// Brake faults section
// Brake cam switch monitoring
TON_1(IN := Lh_off AND Lh_rubbing AND Mode.Brake_maintenance, PT := t#200ms); // TON
TON_2(IN := Rh_off AND Rh_rubbing AND Mode.Brake_maintenance, PT := t#200ms); // TON
cs_Lh_off_before_rubbing := TON_1.Q;
cs_Rh_off_before_rubbing := TON_2.Q;
TON_3(IN := Lh_on AND Lh_rubbing AND Mode.Brake_maintenance, PT := t#200ms); // TON
TON_4(IN := Rh_on AND Rh_rubbing AND Mode.Brake_maintenance, PT := t#200ms); // TON
cs_Lh_on_and_rubbing := TON_3.Q;
cs_Rh_on_and_rubbing := TON_4.Q;
TON_5(IN := Lh_wear AND Lh_on AND Mode.Brake_maintenance, PT := t#200ms); // TON
TON_6(IN := Rh_wear AND Rh_on AND Mode.Brake_maintenance, PT := t#200ms); // TON
cs_Lh_wear_before_on := TON_5.Q;
cs_Rh_wear_before_on := TON_6.Q;
TON_7(IN := Lh_on AND Lh_off AND Mode.Brake_maintenance, PT := t#200ms); // TON
TON_8(IN := Rh_on AND Rh_off AND Mode.Brake_maintenance, PT := t#200ms); // TON
cs_Lh_on_and_off := TON_7.Q;
cs_Rh_on_and_off := TON_8.Q;
TON_9(IN := Lever_on AND Lever_off AND Mode.Brake_maintenance, PT := t#200ms); // TON
TON_10(IN := Lever_on AND Lever_fully_off AND Mode.Brake_maintenance, PT := t#200ms); // TON
cs_Lever_off_and_on := TON_9.Q;
cs_Lever_fully_off_and_on := TON_10.Q;
// Brake lever monitoring
TON_11(IN := Lever_fully_off AND Mode.Manual OR Mode.Auto_go, PT := Off_time); // TON
TON_12(IN := TON_11.Q AND NOT Lh_off AND NOT Trail_brakes AND Clutch.Lh_in AND NOT Lh_test AND Safety.Sc1 AND NOT Mode.Brake_maintenance, PT := t#3s); // TON
cs_Lh_not_fully_off := TON_12.Q;
TON_13(IN := Lever_fully_off AND Mode.Manual OR Mode.Auto_go, PT := Off_time); // TON
TON_14(IN := TON_13.Q AND NOT Rh_off AND NOT Trail_brakes AND Clutch.Rh_in AND NOT Rh_test AND Safety.Sc1 AND NOT Mode.Brake_maintenance, PT := t#3s); // TON
cs_Rh_not_fully_off := TON_14.Q;
TON_15(IN := Lever_on, PT := On_time); // TON
tr_Lh_not_on := TON_15.Q AND NOT Lh_on AND NOT Mode.Brake_maintenance;
// Brake rubbing trips
TON_16(IN := (ABS(Lh_speed)) > Rubbing_speed AND NOT Lh_rubbing AND Safety.Sc1 AND _w1, PT := Rubbing_time); // TON
tr_Lh_rubbing_trip := TON_16.Q;
_w1 := (ABS(Lh_speed)) > 1200 OR TON_17.Q;
TON_17(IN := NOT Trail_brakes, PT := t#1s); // TON
_w3 := TON_17.Q OR _w2;
_w2 := (ABS(Rh_speed)) > 1200;
TON_16(IN := _w3 AND _w4 AND NOT Rh_rubbing AND Safety.Sc1, PT := Rubbing_time); // TON
_w4 := (ABS(Rh_speed)) > Rubbing_speed;
tr_Rh_rubbing_trip := TON_16.Q;
// Brake maintenance trips
tr_No_brake_on_in_maint := Maintenance AND NOT Lh_on AND NOT Rh_on;
tr_Movement_in_maint := Maintenance AND Movement_detect;
tr_Maint_switch_on := NOT (Lh_on OR Rh_on) AND Maintenance_switch;
END_METHOD

END_FUNCTION_BLOCK

// ---- POUs/FBs/FB_Clutch.TcPOU
FUNCTION_BLOCK FB_Clutch
VAR_INPUT
	Lh_in:BOOL; (*Left hand clutch in switch*)
	Lh_out:BOOL; (*Left hand clutch out switch*)
	Rh_in:BOOL; (*Right hand clutch in switch*)
	Rh_out:BOOL; (*Right hand clutch out switch*)
	Lh_movement:BOOL; (*Movement on left hand drum*)
	Rh_movement:BOOL; (*Movement on right hand drum*)
	Lh_raw_depth:DINT; (*Left conveyance raw depth*)
	Rh_raw_depth:DINT; (*Right conveyance raw depth*)
	Allowed_travel_when_out:DINT; (*Amount of travel allowed while engaging/disengaging a clutch*)
END_VAR
VAR_OUTPUT
	tr_Lh_in_and_out:BOOL; (*Left hand clutch in and out switches both energised*)
	tr_Rh_in_and_out:BOOL; (*Right hand clutch in and out switches both energised*)
	tr_Lh_out_movement:BOOL; (*Movement was detected on the left hand drum when the left clutch was out*)
	tr_Rh_out_movement:BOOL; (*Movement was detected on the right hand drum when the right clutch was out*)
	tr_Lh_not_in_movement:BOOL; (*Movement was detected on the left hand drum when the left clutch was not in*)
	tr_Rh_not_in_movement:BOOL; (*Movement was detected on the right hand drum when the right clutch was not in*)
	cs_Too_much_travel_clutching:BOOL; (*There was too much drum travel while engaging/disengaging a clutch*)
	hmi_Status:WORD; (*Status bits for HMI*)
END_VAR
VAR
	TON_0: TON;
	TON_1: TON;
	TON_2: TON;
	TON_3: TON;
	Lh_start_depth: DINT;
	RS_0: RS;
	Rh_start_depth: DINT;
	RS_1: RS;
END_VAR

M_Clutch_data();
M_Clutch_faults();
M_Too_much_travel();

METHOD M_Clutch_data
VAR_INPUT
END_VAR

VAR
	BIT_TO_WORD_V0_0: FB_BIT_TO_WORD_V0;
END_VAR
// Clutch data section
Clutch.Lh_in := Lh_in;
Clutch.Rh_in := Rh_in;
Clutch.Lh_out := Lh_out;
Clutch.Rh_out := Rh_out;
Clutch.Single_drum := Lh_out OR Rh_out;
BIT_TO_WORD_V0_0(bit0 := Lh_in, bit1 := Lh_out, bit2 := Rh_in, bit3 := Rh_out, bit4 := Clutch.Single_drum); // FB_BIT_TO_WORD_V0
hmi_Status := BIT_TO_WORD_V0_0.Word_out;
END_METHOD

METHOD M_Clutch_faults
VAR_INPUT
END_VAR
// Clutch faults section
tr_Lh_in_and_out := Lh_in AND Lh_out;
tr_Rh_in_and_out := Rh_in AND Rh_out;
TON_0(IN := Lh_movement AND Lh_out, PT := t#50ms); // TON
TON_2(IN := Rh_movement AND Rh_out, PT := t#50ms); // TON
tr_Lh_out_movement := TON_0.Q;
tr_Rh_out_movement := TON_2.Q;
TON_1(IN := Lh_movement AND Lh_in, PT := t#50ms); // TON
TON_3(IN := Rh_movement AND Rh_in, PT := t#50ms); // TON
tr_Lh_not_in_movement := TON_1.Q;
tr_Rh_not_in_movement := TON_3.Q;
END_METHOD

METHOD M_Too_much_travel
VAR_INPUT
END_VAR
VAR_INST // added by the converter: edge detectors and wires of the graphical bodies
    _w1, _w3 : ANY;
    _w2, _w4 : DINT;
END_VAR
// Too much travel section
RS_0(SET := ABS(Lh_raw_depth - Lh_start_depth) > Allowed_travel_when_out, RESET1 := _w1); // RS
cs_Too_much_travel_clutching := RS_0.Q1 OR RS_1.Q1;
_w1 := Rh_in OR Rh_out OR Safety.Reset_interlocks;
IF _w1 THEN _w2 := Lh_raw_depth; END_IF
Lh_start_depth := _w2;
RS_1(SET := ABS(Rh_raw_depth - Rh_start_depth) > Allowed_travel_when_out, RESET1 := _w3); // RS
_w3 := Lh_in OR Lh_out OR Safety.Reset_interlocks;
IF _w3 THEN _w4 := Rh_raw_depth; END_IF
Rh_start_depth := _w4;
END_METHOD

END_FUNCTION_BLOCK

// ---- POUs/FBs/FB_Disc_brake.TcPOU
FUNCTION_BLOCK FB_Disc_brake
VAR_INPUT
	S1:REAL; (*Raw analogue value from proxmity transducer in brake caliper module 1*)
	S2:REAL; (*Raw analogue value from proxmity transducer in brake caliper module 2*)
	Pressure:BOOL; (*This input must be active when the pressure is above the threshold used for broken spring detection*)
	Raw_min:REAL; (*Minimum value of raw sensor analogue inputs*)
	Raw_max:REAL; (*Maximum value of raw sensor analogue inputs*)
	Pos_min:REAL; (*Position value corresponding to minimum raw value (typically in mm)*)
	Pos_max:REAL; (*Position value corresponding to maximum raw value (typically in mm)*)
	mA_min:REAL; (*Milliamp value corresponding to minimum raw value (typically 3 to 4mA for 4-20mA transducers)*)
	mA_max:REAL; (*Milliamp value corresponding to maximum raw value (typically 20mA for 4-20mA transducers)*)
	Range_min:REAL; (*Minimum allowed raw value. A lower value will result in an out of range error.*)
	Range_max:REAL; (*Maximum allowed raw value. A lower value will result in an out of range error*)
	Broken_wire:REAL; (*Raw value below which a 4-20mA transducer can be considered open circuit*)
	Off_pos:REAL; (*Position (scaled) value below which the brake module can be considered to be in the "off" position*)
	Rubbing_pos:REAL; (*Position (scaled) value above which the brake module can be considered to be rubbing*)
	On_pos:REAL; (*Average position (scaled) value above which the brake modules can be considered to be "on"*)
	Wear_pos:REAL; (*Average position (scaled) value above which the brake pads can be considered to be "worn"*)
	Speed:REAL;
	Brake_rubbing_speed:REAL;
	Brake_rubbing_on_delay:TIME;
	Colour_scheme:INT; (*An integer value corresponding to the analogue colour scheme to be used on the HMI*)
END_VAR
VAR_OUTPUT
	Pos1:REAL; (*Scaled position value for sensor 1 (typically in mm)*)
	Pos2:REAL; (*Scaled position value for sensor 2 (typically in mm)*)
	mA1:REAL; (*Milliamp value for sensor 1 (for 4-20mA transducers)*)
	mA2:REAL; (*Milliamp value for sensor 2 (for 4-20mA transducers)*)
	Off:BOOL; (*Both brake modules in the "off" position*)
	Rubbing:BOOL; (*At least one of the brake modules is past the "rubbing" position*)
	Brake_on:BOOL; (*The average value of the modules positions is greater than the "on" distance*)
	Wear:BOOL; (*The average value of the modules positions is greater than the "wear" distance*)
	Broken_spring1:BOOL; (*Module 1 has a broken spring (the off position was reached with insufficient pressure)*)
	Broken_spring2:BOOL; (*Module 2 has a broken spring (the off position was reached with insufficient pressure)*)
	S1_out_of_range:BOOL; (*The analogue value of sensor 1 is out of range*)
	S2_out_of_range:BOOL; (*The analogue value of sensor 2 is out of range*)
	S1_broken_wire:BOOL; (*The analogue value of sensor 1 is out of range*)
	S2_broken_wire:BOOL; (*The analogue value of sensor 2 is out of range*)
	tr_Rubbing1:BOOL; (*Side 1 rubbing above allowed speed*)
	tr_Rubbing2:BOOL; (*Side 2 rubbing above allowed speed*)
	HMI1:dut_hmi_Analogue; (*Data structure containing sensor 1 data for HMI*)
	HMI2:dut_hmi_Analogue; (*Data structure containing sensor 2 data for HMI*)
END_VAR
VAR
	Ave_pos:REAL;
	Off1:BOOL;
	Off2:BOOL;
	S1_rubbing:BOOL;
	S2_rubbing:BOOL;
	Raw_to_scaled_0: FB_Raw_to_scaled;
	Raw_to_scaled_1: FB_Raw_to_scaled;
END_VAR

M_Disc_brake_scaling();
M_Disc_brake_positions();
M_Disc_brake_faults();
M_Disc_brake_HMI();

METHOD M_Disc_brake_faults
VAR_INPUT
END_VAR
VAR_INST // added by the converter: edge detectors and wires of the graphical bodies
    _w1, _w2, _w3 : BOOL;
END_VAR
S1_out_of_range := _w1;
S1_broken_wire := _w3 AND NOT Brakes.Maintenance_mode;
S2_out_of_range := (S2 > Range_max OR _w2) AND NOT Brakes.Maintenance_mode;
S2_broken_wire := S2 < Broken_wire AND NOT Brakes.Maintenance_mode;
// Out of range
_w1 := (S1 > Range_max OR S1 < Range_min) AND NOT Brakes.Maintenance_mode;
_w2 := S2 < Range_min;
// Broken wire
_w3 := S1 < Broken_wire;
// Broken spring
Broken_spring1 := (NOT Pressure AND Off1) AND NOT Brakes.Maintenance_mode;
Broken_spring2 := (NOT Pressure AND Off2) AND NOT Brakes.Maintenance_mode;
// Brakes rubbing trip
tr_Rubbing1 := (ABS(Speed)) >= Brake_rubbing_speed AND S1_rubbing;
tr_Rubbing2 := (ABS(Speed)) >= Brake_rubbing_speed AND S2_rubbing;
END_METHOD

METHOD M_Disc_brake_HMI
VAR_INPUT
END_VAR
VAR_INST // added by the converter: edge detectors and wires of the graphical bodies
    _w1, _w2, _w3, _w4, _w8, _w9, _w10, _w12, _w13, _w14, _w15, _w16, _w17 : ANY;
    _w5 : REAL;
    _w6, _w7, _w11 : BOOL;
END_VAR
_w2 := LIMIT(0, _w1, 1000);
_w1 := (Pos2 / (Pos_max - Pos_min)) * 1000;
HMI2.Per_thousand := _w2;
HMI1.Colour := _w3;
HMI1.Colour := _w4;
_w5 := Pos2;
_w7 := _w6;
IF _w7 THEN _w8 := 1; END_IF
HMI2.Colour := _w9;
IF _w7 THEN _w10 := 1; END_IF
HMI2.Colour := _w10;
_w11 := Ave_pos >= Wear_pos;
IF _w11 THEN _w3 := 0; END_IF
IF _w11 THEN _w12 := 0; END_IF
IF Pos1 <= Rubbing_pos THEN _w4 := 3; END_IF
HMI2.Colour := _w12;
HMI2.Value := _w5;
// Pack HMI values into structures. First the scaled values (in correct units), then the percentage values - limited to 0% to 100%.
HMI1.Value := Pos1;
// Set the correct colour for each of the 5 brake positions.
HMI1.Colour := _w13;
HMI1.Colour := 2;
HMI2.Colour := 2;
HMI1.Per_thousand := LIMIT(0, (Pos1 / (Pos_max - Pos_min)) * 1000, 1000);
_w9 := _w14 + HMI2.Colour;
_w6 := Ave_pos >= On_pos;
HMI1.Colour := _w8;
IF Pos2 <= Rubbing_pos THEN _w15 := 3; END_IF
HMI2.Colour := _w15;
IF Pos1 <= Off_pos THEN _w16 := 4; END_IF
IF Pos2 <= Off_pos THEN _w17 := 4; END_IF
HMI1.Colour := _w16;
HMI2.Colour := _w17;
// Offset the colour index according to the colour scheme
_w14 := (Colour_scheme - 1) * 5;
_w13 := _w14 + HMI1.Colour;
END_METHOD

METHOD M_Disc_brake_positions
VAR_INPUT
END_VAR
VAR_INST // added by the converter: edge detectors and wires of the graphical bodies
    _w1, _w2, _w3, _w4, _w5, _w6 : BOOL;
END_VAR
S1_rubbing := _w1;
Off1 := _w2;
_w3 := Pos2 >= Rubbing_pos;
// Brake rubbing
_w2 := Pos1 <= Off_pos;
Rubbing := _w4;
Brake_on := _w5;
Wear := _w6;
// Brake rubbing
_w1 := Pos1 >= Rubbing_pos;
_w4 := _w1 OR _w3;
Off := Off1 AND Off2;
// Brakes on
_w5 := Ave_pos >= On_pos;
// Brake wear
_w6 := Ave_pos >= Wear_pos AND NOT Brakes.Maintenance_mode;
S2_rubbing := _w3;
Off2 := Pos2 <= Off_pos;
END_METHOD

METHOD M_Disc_brake_scaling
VAR_INPUT
END_VAR

VAR
END_VAR
VAR_INST // added by the converter: edge detectors and wires of the graphical bodies
    _w1 : REAL;
END_VAR
Pos1 := Raw_to_scaled_0.Scaled;
Raw_to_scaled_0(
    Value := S2,
    Raw_min := Raw_min,
    Raw_max := Raw_max,
    Scaled_min := Pos_min,
    Scaled_max := Pos_max); // FB_Raw_to_scaled
Pos2 := Raw_to_scaled_0.Scaled;
Raw_to_scaled_1(
    Value := S1,
    Raw_min := Raw_min,
    Raw_max := Raw_max,
    Scaled_min := mA_min,
    Scaled_max := mA_max); // FB_Raw_to_scaled
Ave_pos := _w1;
mA1 := Raw_to_scaled_1.Scaled;
// The raw sensor inputs are scaled to both position and milliamps for fault finding puposes
Raw_to_scaled_0(
    Value := S1,
    Raw_min := Raw_min,
    Raw_max := Raw_max,
    Scaled_min := Pos_min,
    Scaled_max := Pos_max); // FB_Raw_to_scaled
Raw_to_scaled_1(
    Value := S2,
    Raw_min := Raw_min,
    Raw_max := Raw_max,
    Scaled_min := mA_min,
    Scaled_max := mA_max); // FB_Raw_to_scaled
mA2 := Raw_to_scaled_1.Scaled;
_w1 := (Pos1 + Pos2) / 2;
END_METHOD

END_FUNCTION_BLOCK

// ---- POUs/FBs/FB_Raw_to_scaled.TcPOU
FUNCTION_BLOCK FB_Raw_to_scaled
VAR_INPUT
	Value:REAL;
	Raw_min:REAL;
	Raw_max:REAL;
	Scaled_min:REAL;
	Scaled_max:REAL;
END_VAR
VAR_OUTPUT
	Scaled:REAL;
END_VAR
VAR
END_VAR

M_Raw_to_scaled();

METHOD M_Raw_to_scaled
VAR_INPUT
END_VAR
VAR_INST // added by the converter: edge detectors and wires of the graphical bodies
    _w1, _w3 : ANY;
    _w2 : REAL;
END_VAR
_w2 := _w1 + Scaled_min;
_w1 := _w3 * (Scaled_max - Scaled_min);
_w3 := (Value - Raw_min) / Raw_min;
Scaled := _w2;
END_METHOD

END_FUNCTION_BLOCK

// ---- POUs/FBs/FB_Double_drum.TcPOU
FUNCTION_BLOCK FB_Double_drum
VAR_INPUT
	Lh_raw_depth:REAL; (*Raw left hand drum depth*)
	Rh_raw_depth:REAL; (*Raw right hand drum depth*)
	Lh_speed:REAL; (*Left drum speed in mm/s*)
	Rh_speed:REAL; (*Right drum speed in mm/s*)
	Tacho_speed:REAL; (*Tacho speed in mm/s*)
	Speed_ref:REAL; (*Speed reference output to drive in mm/s*)
	Lh_going_up:BOOL; (*Left conveyance moving in the upward direction (forward)*)
	Rh_going_up:BOOL; (*Right conveyance moving in the upward direction (forward)*)
	Lh_movement:BOOL; (*Movement detected on left drum since the brakes were last applied*)
	Rh_movement:BOOL; (*Movement detected on right drum since the brakes were last applied*)
	Enc_xcheck_dist:REAL; (*Allowed variation in the sum of the left and right raw depths since both clutches were put in or a winder reset*)
	Tacho_xcheck_abs:REAL; (*Allowed absolute difference between the tacho speed and encoder speed (added to Tacho_xcheck_percent)*)
	Tacho_xcheck_percent:REAL; (*Allowed percentage difference between the tacho speed and encoder speed (added to Tacho_xcheck_abs)*)
	Speed_ref_xcheck_abs:REAL; (*Allowed absolute difference between the speed reference (delayed) and the encoder speed (added to Speed_ref_xcheck_percent)*)
	Speed_ref_xcheck_percent:REAL; (*Allowed percentage difference between the speed reference (delayed) and the encoder speed (added to Speed_ref_xcheck_abs)*)
	System_response_time:REAL; (*Delay between giving the drive a reference and that speed being reached*)
	Speed_ave_scans:REAL;
END_VAR
VAR_OUTPUT
	Speed:REAL; (*Maximum speed between left and right encoders. Tacho is used if both encoders give zero speed.*)
	Movement:BOOL; (*Movement was detected on the left or right drum since the brakes were last applied*)
	Going_fwd:BOOL; (*The drums are moving in the forward direction*)
	Going_rev:BOOL; (*The drums are moving in the reverse direction*)
	Encoder_sum_xcheck:BOOL; (*The sum of the left and right raw depths has varied more than the allowed amount*)
	Lh_enc_vs_tacho_xcheck:BOOL; (*The difference between the tacho speed and left encoder speed was greater than the allowed amount*)
	Rh_enc_vs_tacho_xcheck:BOOL; (*The difference between the tacho speed and right encoder speed was greater than the allowed amount*)
	Speed_ref_xcheck:BOOL;(*The difference between the speed reference and encoder speed was greater than the allowed amount*)
END_VAR
VAR
	Speed_ref_delay_history:ARRAY[0..100]OF REAL;
	Speed_ref_delayed:REAL;
	System_response_scans:REAL;
	Rh_enc_tacho_diff:REAL;
	Lh_enc_tacho_diff:REAL;
	Speed_ref_diff:REAL;
	Encoder_sum:REAL;
	Required_encoder_sum:REAL;
	Window:REAL;
	F_TRIG_0: F_TRIG;
END_VAR

M_Double_drum_values();
M_Speed_crosschecks();
M_Depth_crosscheck();

METHOD M_Depth_crosscheck
VAR_INPUT
END_VAR
VAR_INST // added by the converter: edge detectors and wires of the graphical bodies
    _w1, _w2 : REAL;
END_VAR
Required_encoder_sum := _w1;
_w2 := Lh_raw_depth + Rh_raw_depth;
// Depth crosscheck between the two encoders
F_TRIG_0(CLK := Brakes.Proved_on); // F_TRIG
Encoder_sum := _w2;
IF F_TRIG_0.Q THEN _w1 := Lh_raw_depth + Rh_raw_depth; END_IF
Encoder_sum := ABS(Required_encoder_sum - Encoder_sum) > Enc_xcheck_dist AND NOT Brakes.Proved_on AND Clutch.Lh_in AND Clutch.Rh_in;
END_METHOD

METHOD M_Double_drum_values
VAR_INPUT
END_VAR
VAR_INST // added by the converter: edge detectors and wires of the graphical bodies
    _w1, _w2, _w3, _w4, _w8, _w9 : BOOL;
    _w5, _w7 : REAL;
    _w6 : ANY;
END_VAR
Going_fwd := _w3;
Going_rev := _w4;
Speed := _w5;
_w7 := SEL(_w6, Rh_speed, -Lh_speed);
_w4 := NOT Going_fwd;
_w6 := (ABS(Lh_speed)) > (ABS(Rh_speed));
// Speed - maximum of the two encoder speeds. If both are zero, use tacho.
_w5 := SEL((ABS(Lh_speed)) < 10 AND _w8 AND _w9, _w7, Tacho_speed);
Movement := _w1 OR _w2;
_w2 := Rh_movement AND Clutch.Rh_in;
_w8 := (ABS(Rh_speed)) < 10;
// Direction
_w3 := SEL(Clutch.Rh_in, Lh_going_up, NOT Rh_going_up);
_w9 := (ABS(Tacho_speed)) > 100;
// Movement detect
_w1 := Lh_movement AND Clutch.Lh_in;
END_METHOD

METHOD M_Speed_crosschecks
VAR_INPUT
END_VAR
VAR
	fbGetCurTaskIdx  : GETCURTASKINDEX;
	nIndex : DINT;
	nUpper : DINT;
	nLower : DINT;
END_VAR
{warning 'TODO: CycleTime here is implicitly converted from UDINT to REAL causing possible data loss.'}
{warning 'TODO: Ive re-written ROL_ARINT, please check @Bret'}
System_response_scans := System_response_time / _TaskInfo[fbGetCurTaskIdx.index].CycleTime;

(* Delay the speed reference to cater for the system response time *)	
//ROL_ARINT(1, Speed_ref_delay_history);

nUpper := UPPER_BOUND(Speed_ref_delay_history, 1);
nIndex := nUpper;

FOR nLower := LOWER_BOUND(Speed_ref_delay_history, 1) TO nUpper DO
	Speed_ref_delay_history[nIndex+1] := Speed_ref_delay_history[nIndex];
	nIndex := nIndex-1;
END_FOR
Speed_ref_delay_history[0] := Speed_ref;
Speed_ref_delayed := Speed_ref_delay_history[System_response_scans];

(* Now crosscheck the speeds. The speed reference will be used as the benchmark because it is the only one guaranteed to be correct. *)
(* The various speed values must agree within a percentage plus a fixed value for low speeds *)

Window := ABS(Speed_ref_delayed) * Tacho_xcheck_percent / 100.0 + Tacho_xcheck_abs;

(* Left encoder vs tacho crosscheck *)
Lh_enc_vs_tacho_xcheck := 0;
IF  Clutch.Lh_in THEN
	Lh_enc_tacho_diff := -Lh_speed - Tacho_speed;
	IF ABS(Lh_enc_tacho_diff) > Window THEN
		Lh_enc_vs_tacho_xcheck := 1;
	END_IF;
END_IF;

(* Right encoder vs tacho crosscheck *)
Rh_enc_vs_tacho_xcheck := 0;
IF Clutch.Rh_in THEN
	Rh_enc_tacho_diff := Rh_speed - Tacho_speed;
	IF ABS(Rh_enc_tacho_diff) > Window THEN
		Rh_enc_vs_tacho_xcheck := 1;
	END_IF;
END_IF;

(* Speed reference vs tacho crosscheck, i.e. speed reference not followed *)

Window := ABS(Speed_ref_delayed) * Speed_ref_xcheck_percent / 100.0 + Speed_ref_xcheck_abs;

Speed_ref_xcheck := 0;
Speed_ref_diff := Speed_ref_delayed - Tacho_speed;
IF ABS(Speed_ref_diff) > Window AND Safety.Sc1 THEN
	Speed_ref_xcheck := 1;
END_IF;
END_METHOD

END_FUNCTION_BLOCK

// ---- POUs/FBs/FB_Drive_control.TcPOU
FUNCTION_BLOCK FB_Drive_control
VAR_INPUT
	Safety_interlock:BOOL;
	Speed:INT; (*When this speed is exceeded, the winder will go from torque control to speed control*)
	Movement_detect:BOOL;
	Motor_fed:BOOL;
	Auto_run:BOOL;
	Auto_ref:INT;
	Auto_trail_brakes:BOOL;
	Speed_scale:INT; (*Full lever speed (modified by creep/slow switch*)
	Lh_allowed_speed:INT;
	Rh_allowed_speed:INT;
	//Current_limit:INT; (*Current limit in Amps*)
	//Max_lever_amps:INT; (*Current ramp rate in Amps*)
	//Speed_ramp_rate:INT; (*Speed ramp rate (accel and decel) in mm/s.*)
	//Current_ramp_rate:INT; (*Ramp rate of armature current reference in A/s used in torque control*)
	Armature_current:REAL; (*Armature current in Amps*)
	Forward_backout:BOOL;
	Reverse_backout:BOOL;
END_VAR
VAR_OUTPUT
	Enable:BOOL; (*Drive enable signal*)
	Start:BOOL; (*Drive start/run signal*)
	Speed_control:BOOL; (*Drive required to be in speed control*)
	Torque_control:BOOL; (*Drive required to be in torque control*)
	Field_weakening:BOOL; (*Field weakening request (for DC drive)*)
	Brake_release:BOOL;
	Trail_brakes:BOOL;
	Driver_ref_final:INT;	
	Torque_prediction:INT;
	Torque_ref:INT; (*Torque reference in amps*)
	Speed_ref:INT; (*Speed reference in mm/s*)
	Drive_speed_ref:REAL; (*Speed reference to drive scaled according to Speed_10V*)
	Drive_torque_ref:INT; (*Torque reference to drive scaled according to Torque_10V (bipolar)*)
	Combined_ref:INT; (*Speed and torque reference combined output (e.g. for TPD32/DCV104)*) 
	cs_No_start:BOOL;
	cs_Stall:BOOL;
	cs_Enable_vs_motor_fed:BOOL;
	hmi_data:dut_hmi_Drive_control;
END_VAR
VAR_IN_OUT
END_VAR
VAR
	R_TRIG_0: R_TRIG;
	RS_0: RS;
	Torq_ctl_brakes_on: BOOL;
	TON_0: TON;
	Kill_torq_ctl: BOOL;
	RS_1: RS;
	RS_2: RS;
	Lincon_0: FB_Lincon;
	Allowed_speed: INT;
	Ref_ramp_0: FB_Ref_ramp;
	Ref_ramp_1: FB_Ref_ramp;
	Torque_prediction_ramp: REAL;
	Lincon_1: FB_Lincon;
	Ref_ramp_2: FB_Ref_ramp;
	Lincon_2: FB_Lincon;
	Lincon_3: FB_Lincon;
	Manual_enable: BOOL;
	Auto_enable: BOOL;
	TON_1: TON;
	Safe_to_lift_brakes: BOOL;
	Lincon_4: FB_Lincon;
	Lincon_5: FB_Lincon;
	Pos_torque: BOOL;
	TON_2: TON;
	RS_3: RS;
	TON_3: TON;
	TON_4: TON;
	TON_5: TON;
	BIT_TO_WORD_V0_0: FB_BIT_TO_WORD_V0;
END_VAR
{warning 'TODO: Remove Combined_ref'}

M_Torque_prediction();
M_Torque_control();
M_Speed_scale();
M_Speed_ref();
M_Torque_ref();
M_Drive_references();
M_Drive_control();
M_Brake_control();
M_Trips();
M_HMI_data();

METHOD M_Brake_control
VAR_INPUT
END_VAR

VAR
END_VAR
VAR_INST // added by the converter: edge detectors and wires of the graphical bodies
    _w1, _w2, _w5, _w6, _w7, _w8, _w9, _w11, _w12, _w13 : BOOL;
    _w3, _w4, _w10 : ANY;
END_VAR
Safe_to_lift_brakes := _w1;
_w3 := TON_2.Q AND _w2;
TON_2(IN := _w4, PT := t#100ms); // TON
_w5 := Armature_current < Lincon_5.Out AND NOT Pos_torque;
_w1 := Safety.Sc1 AND Safety.Sc2 AND Safety.Busc1 AND Safety.Busc2 AND Safety.All_clear;
// Lift the brakes when enough torque has been made or brake lever is released in manual.
Lincon_4(Enable := 1, Input := Torque_prediction, Multiplier := 80, Divisor := 100, Offset := -100); // LINCON
_w4 := _w6 OR Brake_release OR _w5;
_w6 := Armature_current > Lincon_4.Out AND Pos_torque;
_w2 := Auto_run OR _w7;
Lincon_5(Enable := 1, Input := Torque_prediction, Multiplier := 80, Divisor := 100, Offset := -100); // LINCON
_w10 := _w8 AND NOT _w9 AND NOT Brakes.Lever_on AND Safety.All_clear AND NOT Mode.Auto AND Mode.Manual;
_w11 := (ABS(Speed)) <= sp.Drive.Brake_apply_speed;
_w8 := Motor_fed OR Brakes.Maintenance_mode;
_w7 := Auto_run AND _w10;
_w9 := Mode.Manual AND Mode.Single_lever_control AND NOT Power_lever.Button AND Power_lever.Neutral AND _w11;
_w12 := _w3 OR _w10 AND (NOT Mode.Single_lever_control OR Brakes.Lh_test OR Brakes.Rh_test) AND NOT Auto_run;
RS_3(SET := _w11 AND Safety.Control_stop, RESET1 := NOT Safety.Control_stop); // RS
Brake_release := _w13;
_w13 := _w12 AND NOT (NOT RS_3.Q1);
// Enable trail brakes when requested in auto mode. De-energise the valve when the brakes are on.
Trail_brakes := Auto_trail_brakes;
END_METHOD

METHOD M_Drive_control
VAR_INPUT
END_VAR

VAR
END_VAR
VAR_INST // added by the converter: edge detectors and wires of the graphical bodies
    _w1, _w2, _w3, _w4, _w5, _w7, _w8, _w9, _w10, _w11 : BOOL;
    _w6 : ANY;
END_VAR
// Auto mode
_w1 := NOT Brakes.Proved_on_500ms AND Auto_enable;
_w3 := _w2 AND Mode.Auto AND Safety_interlock;
// Speed control
_w4 := Enable AND NOT Torque_control;
Enable := _w5;
// Start drive
Start := Enable;
TON_1(IN := _w6, PT := t#5s); // TON
_w5 := _w7 AND NOT Brakes.Maintenance_mode;
_w2 := _w1 OR _w8;
Auto_enable := _w3;
// Manual mode
_w10 := _w9 AND Mode.Manual AND Safety_interlock;
_w9 := NOT Brakes.Proved_on_500ms AND Manual_enable OR _w11;
Manual_enable := _w10;
_w11 := Torque_control OR NOT Brakes.Lever_on OR NOT Power_lever.Neutral;
_w8 := Auto_run AND NOT Safety.Control_stop;
// Enable output
_w7 := Manual_enable OR Auto_enable;
Speed_control := _w4;
// Field weakening (for DC machines)
_w6 := Enable AND NOT Torque_control;
Field_weakening := TON_1.Q;
END_METHOD

METHOD M_Drive_references
VAR_INPUT
END_VAR

VAR
	Drive_abs_torque: REAL;
	Pos_torque: BOOL;
END_VAR
VAR_INST // added by the converter: edge detectors and wires of the graphical bodies
    _w1 : INT;
    _w2 : REAL;
END_VAR
Drive_speed_ref := Lincon_2.Out;
Lincon_3(
    Enable := 1,
    Input := ABS(Torque_ref),
    Multiplier := 10000,
    Divisor := sp.Drive.Max_drive_torque,
    Offset := 0); // FB_Lincon
Drive_abs_torque := Lincon_3.Out;
Drive_torque_ref := _w1;
_w2 := SEL(Torque_control, Drive_speed_ref, Drive_torque_ref);
Lincon_2(
    Enable := 1,
    Input := Speed_ref,
    Multiplier := 10000,
    Divisor := sp.Drive.Max_drive_speed,
    Offset := 0); // FB_Lincon
Combined_ref := _w2;
Pos_torque := Torque_ref >= 0;
_w1 := SEL(Pos_torque, -1, 1) * Drive_abs_torque;
END_METHOD

METHOD M_HMI_data
VAR_INPUT
END_VAR
hmi_data.Torque_ref := Torque_prediction;
hmi_data.Speed_ref := Speed_ref;
hmi_data.Torque_ref := Torque_ref;
BIT_TO_WORD_V0_0(
    bit0 := Enable,
    bit1 := Manual_enable,
    bit2 := Auto_enable,
    bit3 := Torque_control,
    bit4 := Speed_control,
    bit5 := Field_weakening,
    bit6 := Brake_release,
    bit7 := Trail_brakes,
    bit8 := Auto_run,
    bit9 := Motor_fed); // FB_BIT_TO_WORD_V0
hmi_data.Status := BIT_TO_WORD_V0_0.Word_out;
END_METHOD

METHOD M_Speed_ref
VAR_INPUT
END_VAR

VAR
	
END_VAR
VAR_INST // added by the converter: edge detectors and wires of the graphical bodies
    _w1, _w3, _w4, _w5, _w6, _w7 : ANY;
    _w2 : INT;
END_VAR
_w2 := SEL(Clutch.Rh_in, Lh_allowed_speed, _w1);
_w1 := SEL(Clutch.Lh_in, Rh_allowed_speed, _w3);
Allowed_speed := _w2;
// Speed ref section
// Apply allowed speed according to clutch states
_w3 := MIN(Lh_allowed_speed, Rh_allowed_speed);
_w7 := SEL(Safety.Control_stop, _w6, 0);
// Ramp speed reference according to ramp_rate
_w6 := SEL(Mode.Auto AND Auto_run, Driver_ref_final, Auto_ref);
Speed_ref := MIN(MAX(Ref_ramp_0.Speed_ref, _w4), _w5);
Ref_ramp_0(
    Speed_req_in := _w7,
    Allowed_speed := Allowed_speed,
    Rate := Speed_ramp_rate,
    Zero := NOT Safety_interlock OR Brakes.Proved_on OR Torque_control,
    S_Func_scans := sp.Drive.Speed_S_func_scans); // FB_Ref_ramp
_w4 := SEL(Forward_backout, -32767, sp.Drive.Backout_min_speed);
_w5 := SEL(Reverse_backout, 32767, sp.Drive.Backout_min_speed);
END_METHOD

METHOD M_Speed_scale
VAR_INPUT
END_VAR
// Speed scale section
Driver_ref_final := Power_lever.Cubic;
// In manual mode, rescale drivers lever according to speed selection switches
IF NOT (NOT Mode.Auto) THEN
    Lincon_0(
        Enable := NOT (NOT Mode.Auto),
        Input := Driver_ref_final,
        Multiplier := Speed_scale,
        DIvisor := 10000,
        Offset := 0); // FB_Lincon
END_IF
Driver_ref_final := Lincon_0.Out;
END_METHOD

METHOD M_Torque_control
VAR_INPUT
END_VAR
VAR_INST // added by the converter: edge detectors and wires of the graphical bodies
    _w1, _w2, _w3, _w4, _w5, _w6, _w7 : BOOL;
END_VAR
// Torque control section
// Kill torque control when brake lever is put back on or power lever returns to neutral before brake lever is released.
R_TRIG_0(CLK := Brakes.Lever_on); // R_TRIG
RS_0(SET := R_TRIG_0.Q, RESET1 := Torque_control); // RS
Torq_ctl_brakes_on := RS_0.Q1;
TON_0(IN := (Mode.Auto OR Brakes.Lever_on) AND Power_lever.Neutral AND Torque_control OR Torq_ctl_brakes_on, PT := t#500ms); // TON
Kill_torq_ctl := TON_0.Q;
// Torque control logic
Torque_control := (((Torque_control OR Power_lever.Neutral) AND Kill_torq_ctl OR NOT Brakes.Lever_on OR _w1) AND Mode.Manual OR _w2) AND Safety_interlock AND _w3 AND _w4;
_w2 := Auto_run AND Mode.Auto;
_w1 := (ABS(Armature_current)) > 100 AND _w5;
RS_2(SET := Brakes.Lh_test AND NOT Enable, RESET1 := NOT Brakes.Lh_test); // RS
// Kick out of torque
// control after time-out
_w3 := RS_2.Q1 OR RS_2.Q1 OR _w6;
_w5 := Brakes.Lh_test OR Brakes.Rh_test;
RS_2(SET := Brakes.Rh_test AND NOT Enable, RESET1 := NOT Brakes.Rh_test); // RS
RS_1(SET := (ABS(Speed)) > sp.Drive.Torque_ctrl_max_speed, RESET1 := Brakes.Proved_on_500ms); // RS
_w6 := RS_1.Q1 AND Movement_detect;
_w4 := NOT (Auto_run AND Auto_trail_brakes AND NOT Brakes.Lh_on OR Brakes.Lh_off) AND Clutch.Lh_in OR _w7;
_w7 := NOT (Auto_run AND Auto_trail_brakes AND NOT Brakes.Rh_on OR Brakes.Rh_off) AND Clutch.Rh_in;
END_METHOD

METHOD M_Torque_prediction
VAR_INPUT
END_VAR
{warning 'TODO: Lead Lag Filter needs to be made to work correctly.'}
VAR_INST // added by the converter: edge detectors and wires of the graphical bodies
    _w1, _w2, _w4, _w5, _w12, _w13, _w14, _w15, _w17, _w18, _w19, _w20 : ANY;
    _w3, _w6, _w7, _w8, _w9, _w10, _w11 : BOOL;
    _w16 : INT;
END_VAR
// note: this text did not pass the execution check against the stored diagram
_w4 := _w3 AND FB_LAG_FILTER_0.Out AND SEL(_w1, _w2, -Dynamic_friction_current);
_w3 := SEL(Enable, 0, _w5);
_w5 := _w6 AND _w7 AND _w8 AND _w9 AND _w10 AND _w11;
_w7 := SEL(Clutch.Rh_in, 0, -sp.Drive.Rh_cage_mass_current);
Torque_prediction := _w4;
_w8 := SEL(Clutch.Lh_in, 0, _w12);
_w9 := SEL(Clutch.Rh_in, 0, _w13);
_w13 := (Rh_rope_mass_current * Rh_depth) / Levels[Bottom_level];
_w15 := SEL(Lh_half_load, _w14, Full_payload_current/2);
// Now add/subtract the currents required to hold each cage at the bank in single drum.
// Note: All torque values have units of Amps.
_w6 := SEL(Clutch.Lh_in, 0, sp.Drive.Lh_cage_mass_current);
_w16 := Speed_ref;
Speed_ramp_rate := _w17;
FB_LAG_FILTER_0(In := _w18, Time_const := Accel_torque_lag); // FB_Lag_filter
_w18 := Speed_ramp_rate * A_s2_per_m;
// Now add/subtract the pro rata out of balance currents.
_w12 := (Lh_rope_mass_current * Lh_depth) / Levels[Bottom_level];
// Cage payload current
_w14 := SEL(Lh_full_load, 0, Full_payload_current);
_w10 := SEL(Mode.Auto, _w15, 0);
_w11 := SEL(Mode.Auto, _w19, 0);
_w19 := SEL(Rh_half_load, _w20, Full_payload_current/2);
_w20 := SEL(Rh_full_load, 0, Full_payload_current);
_w2 := SEL(Speed_ref > 0, 0, Dynamic_friction_current);
// Acceleration torque current
_w17 := (Speed_ref - Speed_ref_prev) / _TaskInfo[1].CycleTime;
Speed_ref_prev := _w16;
// Current to overcome dynamic friction
_w1 := Speed_ref < 0;
// ???: input not connected
END_METHOD

METHOD M_Torque_ref
VAR_INPUT
END_VAR

VAR
END_VAR
VAR_INST // added by the converter: edge detectors and wires of the graphical bodies
    _w1 : INT;
    _w2, _w3, _w4, _w6, _w7, _w9, _w10 : ANY;
    _w5, _w8 : BOOL;
END_VAR
Torque_ref := _w1;
_w1 := SEL(Safety_interlock, 0, _w2);
_w4 := _w3 * 100.0;
// Ramp the torque prediction in and out
_w5 := Brakes.Proved_on AND NOT Auto_run;
Ref_ramp_1(
    Speed_req_in := _w6,
    Allowed_speed := Current_limit,
    Rate := Current_ramp_rate,
    S_Func_scans := sp.Drive.Current_S_func_scans); // FB_Ref_ramp
_w6 := SEL(_w5, sp.Drive.Max_drive_torque, 0);
Torque_prediction_ramp := Ref_ramp_1.Speed_ref;
// Add manual reference to predicted current when in manual mode
_w3 := Power_lever.Linear * Max_lever_amps;
Ref_ramp_2(
    Speed_req_in := _w4,
    Allowed_speed := Current_limit,
    Rate := Current_ramp_rate,
    Zero := _w7,
    S_Func_scans := sp.Drive.Current_S_func_scans); // FB_Ref_ramp
_w7 := Mode.Manual AND Power_lever.Neutral OR Mode.Auto OR NOT Torque_control OR _w8;
_w8 := Mode.Single_lever_control AND Brakes.Lh_test AND Brakes.Lh_test;
_w2 := LIMIT(-Current_limit, Ref_ramp_2.Speed_ref + _w9, Current_limit);
_w9 := SEL(Brakes.Lh_test OR Brakes.Rh_test, _w10, 0);
_w10 := LIMIT(-Torque_prediction_ramp, Torque_prediction, Torque_prediction_ramp);
END_METHOD

METHOD M_Trips
VAR_INPUT
END_VAR
VAR_INST // added by the converter: edge detectors and wires of the graphical bodies
    _w1, _w3, _w5 : BOOL;
    _w2, _w4 : ANY;
END_VAR
No_start := TON_3.Q;
Enable_vs_motor_fed := TON_5.Q;
_w2 := Brakes.Lever_on OR _w1 OR Brakes.Rh_on AND Clutch.Rh_in;
// No start trip
_w1 := Brakes.Lh_on AND Clutch.Lh_in;
TON_3(IN := _w2 AND Enable, PT := sp.Drive.No_start_time); // TON
// Stall trip
_w3 := (ABS(Speed_ref)) < sp.Drive.Stall_speed;
TON_4(IN := _w4, PT := sp.Drive.Stall_time); // TON
Stall := TON_4.Q;
_w4 := _w3 AND Enable AND NOT Brakes.Lever_on AND NOT Brakes.Lh_test AND NOT Brakes.Rh_test AND _w5;
_w5 := (ABS(Armature_current)) > sp.Drive.Stall_current;
// Motor fed crosscheck with PLC enable
TON_5(IN := Motor_fed XOR Enable, PT := sp.Drive.Motor_fed_delay); // TON
END_METHOD

END_FUNCTION_BLOCK

// ---- POUs/FBs/FB_Lincon.TcPOU
FUNCTION_BLOCK FB_Lincon
VAR_INPUT
	Enable:BOOL; (**)
	Input:REAL; (**)
	Multiplier:REAL; (**)
	Divisor:REAL; (**)
	Offset:REAL; (**)
END_VAR
VAR_OUTPUT
	Out:REAL; (**)
END_VAR
VAR
END_VAR
VAR
	Mul_r:REAL;
	Div_r:REAL;
	In_r:REAL;
	Out_r:REAL;
	Err_b:BOOL;
	tempMemAddr:REAL;
END_VAR

{warning 'TODO: Two places need the equivalent of %S18 placed here. Be sure to delete the tempMemAddr var when you are done.'}
VAR // added by the converter: edge detectors and wires of the graphical bodies
    _w1, _w2, _w9, _w11, _w12, _w13, _w15 : BOOL;
    _w3, _w4, _w5, _w6, _w7, _w8, _w14 : REAL;
    _w10, _w16 : ANY;
END_VAR

// This function block used the formula : Output = Input * multiplier/divisor + offset
IF Enable THEN _w1 := Divisor <> 0.0; END_IF
_w2 := _w1;
IF _w2 THEN _w3 := Input * Multiplier; END_IF
Out := _w4;
IF _w2 THEN _w4 := _w3 / Divisor; END_IF
Out := _w5;
// Need to add %S18 here
tempMemAddr := _w6;
IF _w1 THEN _w7 := Out + Offset; END_IF
IF Enable THEN _w8 := _w7; END_IF
Out := _w8;
IF _w9 THEN _w10 := -32768; END_IF
_w11 := Enable;
IF _w11 THEN (* Divisor = 0.0; result not used *) END_IF
Out := _w10;
_w12 := _w1 AND tempMemAddr;
Err_b := _w12;
// Need to add %S18 here
_w13 := _w12;
IF _w13 THEN _w14 := Out + Offset; END_IF
IF _w13 THEN _w15 := _w14 > 32767; END_IF
IF _w15 THEN _w5 := 32767; END_IF
IF _w13 THEN _w9 := _w14 < -32768; END_IF
IF _w11 THEN _w16 := 0; END_IF
Out := _w16;
IF Err_b THEN _w6 := 0.0; END_IF

END_FUNCTION_BLOCK

// ---- POUs/FBs/FB_Ref_ramp.TcPOU
FUNCTION_BLOCK FB_Ref_ramp
VAR_INPUT
	Speed_req_in:REAL;
	Allowed_speed:REAL;
	Rate:REAL;
	Zero:BOOL;
	S_Func_scans:REAL;
END_VAR
VAR_OUTPUT
	Speed_ref:INT;
END_VAR
VAR
	Speed_req_real: REAL;
	Speed_step: REAL;
	Speed_ref_real: REAL;
	Speed_up: BOOL;
	FB_CTRL_MOVING_AVERAGE_0: FB_CTRL_MOVING_AVERAGE;
END_VAR
{warning 'TODO: Moving average FB needs to be set up by Bret'}
VAR // added by the converter: edge detectors and wires of the graphical bodies
    _w1, _w3, _w6, _w7 : ANY;
    _w2 : BOOL;
    _w4, _w5, _w8, _w9 : REAL;
END_VAR

Speed_req_real := LIMIT(_w1, Speed_req_in, Allowed_speed);
Speed_up := _w2;
// Apply S-function and zero the output when required
IF Zero THEN _w3 := 0; END_IF
// Speed ramp section
// Calculate speed change required per scan
_w4 := Rate * 0;
Speed_step := _w5;
IF NOT Speed_up THEN _w7 := LIMIT(Speed_req_real, _w6, 100000); END_IF
// This input was %SW0 and needs to be addressed properly here
// Make sure the speed reference is never greater than the maximum allowed speed.
_w1 := 0 - Allowed_speed;
Speed_ref_real := _w3;
_w5 := _w4 / 1000;
Speed_ref_real := _w8;
Speed_ref_real := _w7;
// Determine whether the speed step needs to be added or subtracted.
_w2 := Speed_req_real > Speed_ref_real;
IF NOT Speed_up THEN _w6 := Speed_ref_real - Speed_step; END_IF
// Add/subtract the speed step and make sure it doesn't go past the requested speed.
IF Speed_up THEN _w9 := Speed_ref_real + Speed_step; END_IF
IF Speed_up THEN _w8 := LIMIT(-100000, _w9, Speed_req_real); END_IF
FB_CTRL_MOVING_AVERAGE_0(); // FB_CTRL_MOVING_AVERAGE

END_FUNCTION_BLOCK

// ---- POUs/FBs/FB_Encoder_depth.TcPOU
FUNCTION_BLOCK FB_Encoder_depth
VAR_INPUT
	Count:REAL;
	mm_per_count:REAL;
	Rope_capping_mode:BOOL;
	Calibrate:BOOL;
	Cal_switch_depth:REAL;
	Cal_window_up:REAL;
	Cal_window_down:REAL;
	Manual_cal:BOOL;
	Manual_cal_depth:REAL;
	Roll_over_count:REAL;
	Reset_offset:BOOL;
	Speed_ave_intervals:REAL;
	Scans_per_update:REAL;
	Brakes_proved_on:BOOL;
	Winder_reset:BOOL;
	Min_depth:REAL;
	Max_depth:REAL;
	Wind_top_depth:REAL;
	Wind_bottom_depth:REAL;
	Mid_wind_error:REAL;
	Direction_hysteresis:REAL;
	Movement_detect_dist:REAL;
END_VAR
VAR_OUTPUT
	Raw_depth:REAL;
	Calibrated_depth:REAL;
	Compensated_depth:REAL;
	Offset:REAL;
	Speed:REAL;
	New_depth:BOOL;
	Going_up:BOOL;
	Movement_detect:BOOL;
	Depth_out_of_range:BOOL;
	Offset_out_of_range:BOOL;
	Closed_above:BOOL;
	Open_below:BOOL;
	Raw_count:REAL;
	Corrected_count:REAL;
END_VAR
VAR_IN_OUT
	hmi_data:dut_hmi_Depth;
	Zero_count:REAL;
	Depth_history:ANY_ARRAY_REAL;
END_VAR
VAR
	Encoder_mm:REAL;
	Captured_depth:REAL;
	Disallow_multiple_cal:BOOL;
	Raw_depth_prev:REAL;
	Scan_count:REAL;
	Late_depth:BOOL;
	Brakes_on_depth:REAL;
	Brakes_proved_on_500ms:BOOL;
	Compensation:REAL;
	Max_pos_reached:REAL;
	hmi_Manual_cal:BOOL;
	Zero_depth_count:REAL;
	FB_WORD_TO_BIT_V0_0: FB_WORD_TO_BIT_V0;
	R_TRIG_0: R_TRIG;
	R_TRIG_1: R_TRIG;
	F_TRIG_0: F_TRIG;
	RS_0: RS;
	TON_0: TON;
	R_TRIG_2: R_TRIG;
	RS_1: RS;
	SR_0: SR;
	FB_BIT_TO_WORD_V0_0: FB_BIT_TO_WORD_V0;
END_VAR

M_HMI_command();
M_Corrected_count();
M_Encoder_depth();
M_Layering_compensation();
M_Encoder_cal();
M_Depth_history();
M_Speed();
M_Movement_detect();
M_Direction();
M_HMI_data();

METHOD M_Corrected_count
VAR_INPUT
END_VAR
{warning 'TODO: THe last two FBs in this method seem incomplete - no output!'}
VAR_INST // added by the converter: edge detectors and wires of the graphical bodies
    _w1, _w2 : REAL;
    _w3 : BOOL;
END_VAR
